# EPICS substitutions: elioApp/Db/EL4134.substitutions
file EL4134.template { pattern
{ CHAN	}
{ 1	}
{ 2	}
{ 3	}
{ 4	}
}
